{attribute 'qualified_only'}
{attribute 'strict'}
TYPE CalibStateType :
(
	PRE_LAUNCH := 0, // When the user is inputting settings. 
	TEST_SETUP := 1, // When the automation is getting the test ready
	TEST_ACTIVE := 2, // When the test is actively running. 
	TEST_FINISHED := 3, // When all calibration rounds have been completed. 
	ABORT := -1 // When the user has interrupted a test. 
	
);
END_TYPE

(* stored: Version 1.1.0.1, ProductVersion 3.1.4024.12
   DUT CalibStateType: Id {d8c2773c-e73d-4d5a-9f38-136029e63922} *)
